// TIA Portal V17 export
// export: Created 2025-03-20T13:42:36.7741063Z, ExportSetting WithDefaults, DisplayName Totally Integrated Automation Portal, DisplayVersion V17 Update 8, DisplayName TIA Portal Openness, DisplayVersion V17 Update 8, DisplayName TIA Portal Version Control Interface, DisplayVersion V17, DisplayName SINAMICS Startdrive Advanced, DisplayVersion V17 SP2, DisplayName SINAMICS Startdrive G110M, G120, G120C, G120D, G120P, G115D, DisplayVersion V17 SP2, DisplayName SINAMICS Startdrive G130, G150, S120, S150, SINAMICS MV, S210, DisplayVersion V17 SP2, DisplayName STEP 7 Professional, DisplayVersion V17 Update 8, DisplayName SINUMERIK ONE STEP 7 Toolbox, DisplayVersion V17 Update 12, DisplayName SINUMERIK 840D sl STEP 7 Toolbox, DisplayVersion V17 Update 12, DisplayName STEP 7 Safety, DisplayVersion V17 Update 6, DisplayName WinCC Advanced, DisplayVersion V17 Update 8
FUNCTION "FC1302_UNIT_03_STATION_0_CYCLE" : Void   // FC1302, LAD
{ S7_Optimized_Access := 'FALSE' }
AUTHOR : ETXETAR
VERSION : 1.0
// stored: AutoNumber false, IsIECCheckEnabled false, SetENOAutomatically false, UDAEnableTagReadback false
   VAR CONSTANT
      FC_NUMBER : DInt := 1302;
   END_VAR
   VAR_TEMP   // added for the SCL form of the ladder/FBD networks
      _w1 : Bool;
   END_VAR
BEGIN

REGION Network 1: GENERAL CONDITIONS
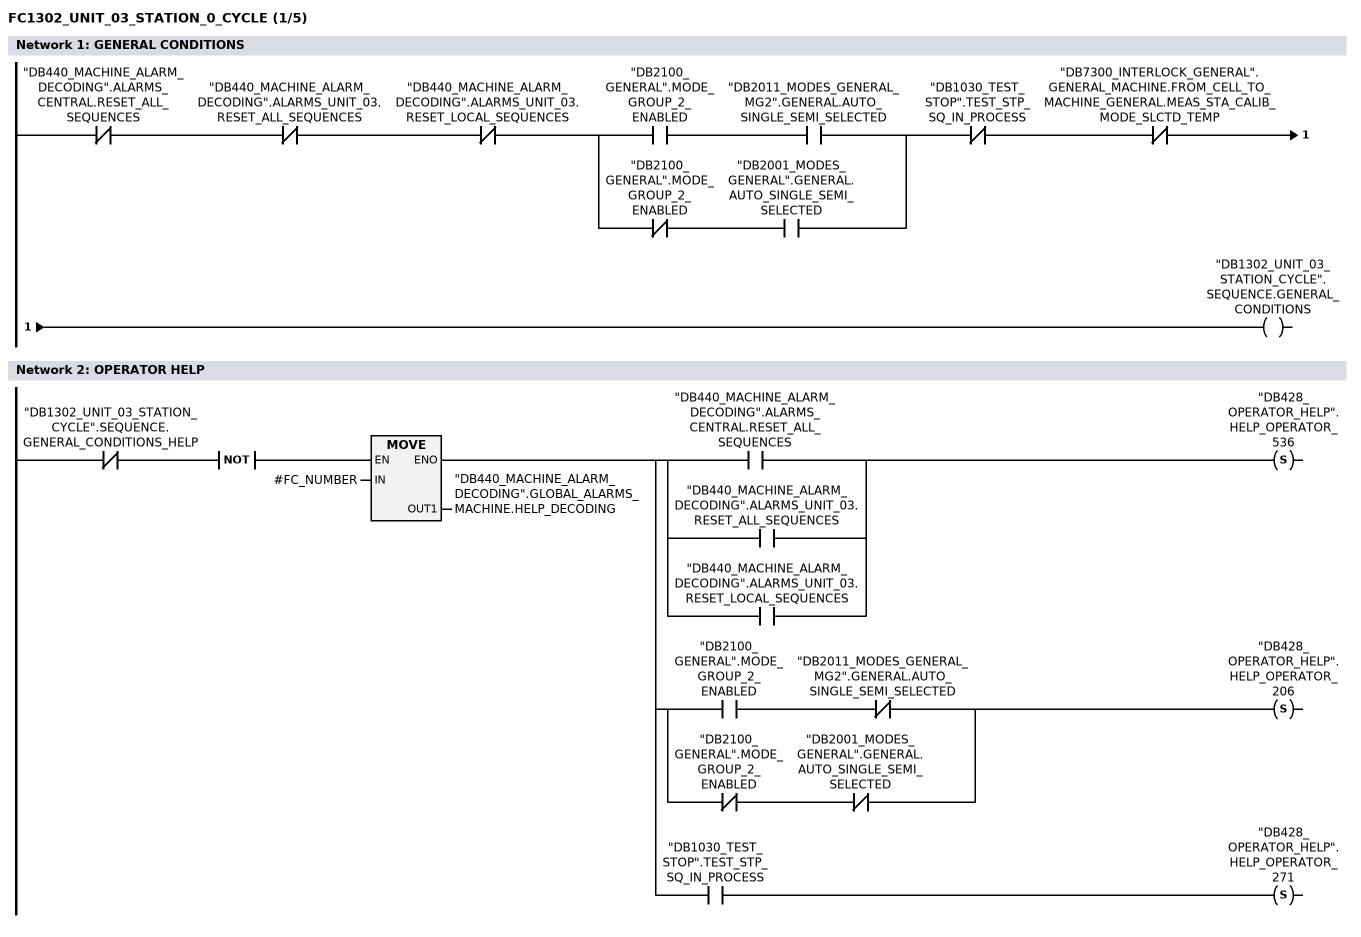
   RUNG wire#powerrail
      I_Contact( "DB440_MACHINE_ALARM_DECODING".ALARMS_CENTRAL.RESET_ALL_SEQUENCES )
      I_Contact( "DB440_MACHINE_ALARM_DECODING".ALARMS_UNIT_03.RESET_ALL_SEQUENCES )
      I_Contact( "DB440_MACHINE_ALARM_DECODING".ALARMS_UNIT_03.RESET_LOCAL_SEQUENCES )
      wire#w1
      Contact( "DB2100_GENERAL".MODE_GROUP_2_ENABLED )
      Contact( "DB2011_MODES_GENERAL_MG2".GENERAL.AUTO_SINGLE_SEMI_SELECTED )
      wire#w2
      I_Contact( "DB1030_TEST_STOP".TEST_STP_SQ_IN_PROCESS )
      I_Contact( "DB7300_INTERLOCK_GENERAL".GENERAL_MACHINE.FROM_CELL_TO_MACHINE_GENERAL.MEAS_STA_CALIB_MODE_SLCTD_TEMP )
      Coil( "DB1302_UNIT_03_STATION_CYCLE".SEQUENCE.GENERAL_CONDITIONS )
   END_RUNG
   RUNG wire#w1
      I_Contact( "DB2100_GENERAL".MODE_GROUP_2_ENABLED )
      Contact( "DB2001_MODES_GENERAL".GENERAL.AUTO_SINGLE_SEMI_SELECTED )
   END_RUNG wire#w2
   // the same network as SCL:
   "DB1302_UNIT_03_STATION_CYCLE".SEQUENCE.GENERAL_CONDITIONS := NOT "DB440_MACHINE_ALARM_DECODING".ALARMS_CENTRAL.RESET_ALL_SEQUENCES AND NOT "DB440_MACHINE_ALARM_DECODING".ALARMS_UNIT_03.RESET_ALL_SEQUENCES AND NOT "DB440_MACHINE_ALARM_DECODING".ALARMS_UNIT_03.RESET_LOCAL_SEQUENCES AND (("DB2100_GENERAL".MODE_GROUP_2_ENABLED AND "DB2011_MODES_GENERAL_MG2".GENERAL.AUTO_SINGLE_SEMI_SELECTED) OR (NOT "DB2100_GENERAL".MODE_GROUP_2_ENABLED AND "DB2001_MODES_GENERAL".GENERAL.AUTO_SINGLE_SEMI_SELECTED)) AND NOT "DB1030_TEST_STOP".TEST_STP_SQ_IN_PROCESS AND NOT "DB7300_INTERLOCK_GENERAL".GENERAL_MACHINE.FROM_CELL_TO_MACHINE_GENERAL.MEAS_STA_CALIB_MODE_SLCTD_TEMP;
END_REGION

REGION Network 2: OPERATOR HELP
   RUNG wire#powerrail
      I_Contact( "DB1302_UNIT_03_STATION_CYCLE".SEQUENCE.GENERAL_CONDITIONS_HELP )
      Not()
      { S7_GenerateENO := "TRUE" } Move(in := #FC_NUMBER, out1 => "DB440_MACHINE_ALARM_DECODING".GLOBAL_ALARMS_MACHINE.HELP_DECODING)
      wire#w1
      Contact( "DB440_MACHINE_ALARM_DECODING".ALARMS_CENTRAL.RESET_ALL_SEQUENCES )
      wire#w2
      S_Coil( "DB428_OPERATOR_HELP".HELP_OPERATOR_536 )
   END_RUNG
   RUNG wire#w1
      Contact( "DB440_MACHINE_ALARM_DECODING".ALARMS_UNIT_03.RESET_ALL_SEQUENCES )
   END_RUNG wire#w2
   RUNG wire#w1
      Contact( "DB440_MACHINE_ALARM_DECODING".ALARMS_UNIT_03.RESET_LOCAL_SEQUENCES )
   END_RUNG wire#w2
   RUNG wire#w1
      Contact( "DB2100_GENERAL".MODE_GROUP_2_ENABLED )
      I_Contact( "DB2011_MODES_GENERAL_MG2".GENERAL.AUTO_SINGLE_SEMI_SELECTED )
      wire#w3
      S_Coil( "DB428_OPERATOR_HELP".HELP_OPERATOR_206 )
   END_RUNG
   RUNG wire#w1
      I_Contact( "DB2100_GENERAL".MODE_GROUP_2_ENABLED )
      I_Contact( "DB2001_MODES_GENERAL".GENERAL.AUTO_SINGLE_SEMI_SELECTED )
   END_RUNG wire#w3
   RUNG wire#w1
      Contact( "DB1030_TEST_STOP".TEST_STP_SQ_IN_PROCESS )
      S_Coil( "DB428_OPERATOR_HELP".HELP_OPERATOR_271 )
   END_RUNG
   // the same network as SCL:
   // ENO of a box is taken as its EN; it also drops when the box reports an error
   #_w1 := NOT (NOT "DB1302_UNIT_03_STATION_CYCLE".SEQUENCE.GENERAL_CONDITIONS_HELP);
   IF #_w1 THEN "DB440_MACHINE_ALARM_DECODING".GLOBAL_ALARMS_MACHINE.HELP_DECODING := #FC_NUMBER; END_IF;
   IF #_w1 AND ("DB440_MACHINE_ALARM_DECODING".ALARMS_CENTRAL.RESET_ALL_SEQUENCES OR "DB440_MACHINE_ALARM_DECODING".ALARMS_UNIT_03.RESET_ALL_SEQUENCES OR "DB440_MACHINE_ALARM_DECODING".ALARMS_UNIT_03.RESET_LOCAL_SEQUENCES) THEN
       "DB428_OPERATOR_HELP".HELP_OPERATOR_536 := TRUE;
   END_IF;
   IF #_w1 AND (("DB2100_GENERAL".MODE_GROUP_2_ENABLED AND NOT "DB2011_MODES_GENERAL_MG2".GENERAL.AUTO_SINGLE_SEMI_SELECTED) OR (NOT "DB2100_GENERAL".MODE_GROUP_2_ENABLED AND NOT "DB2001_MODES_GENERAL".GENERAL.AUTO_SINGLE_SEMI_SELECTED)) THEN
       "DB428_OPERATOR_HELP".HELP_OPERATOR_206 := TRUE;
   END_IF;
   IF #_w1 AND "DB1030_TEST_STOP".TEST_STP_SQ_IN_PROCESS THEN
       "DB428_OPERATOR_HELP".HELP_OPERATOR_271 := TRUE;
   END_IF;
END_REGION

REGION Network 3: INITIAL CONDITIONS
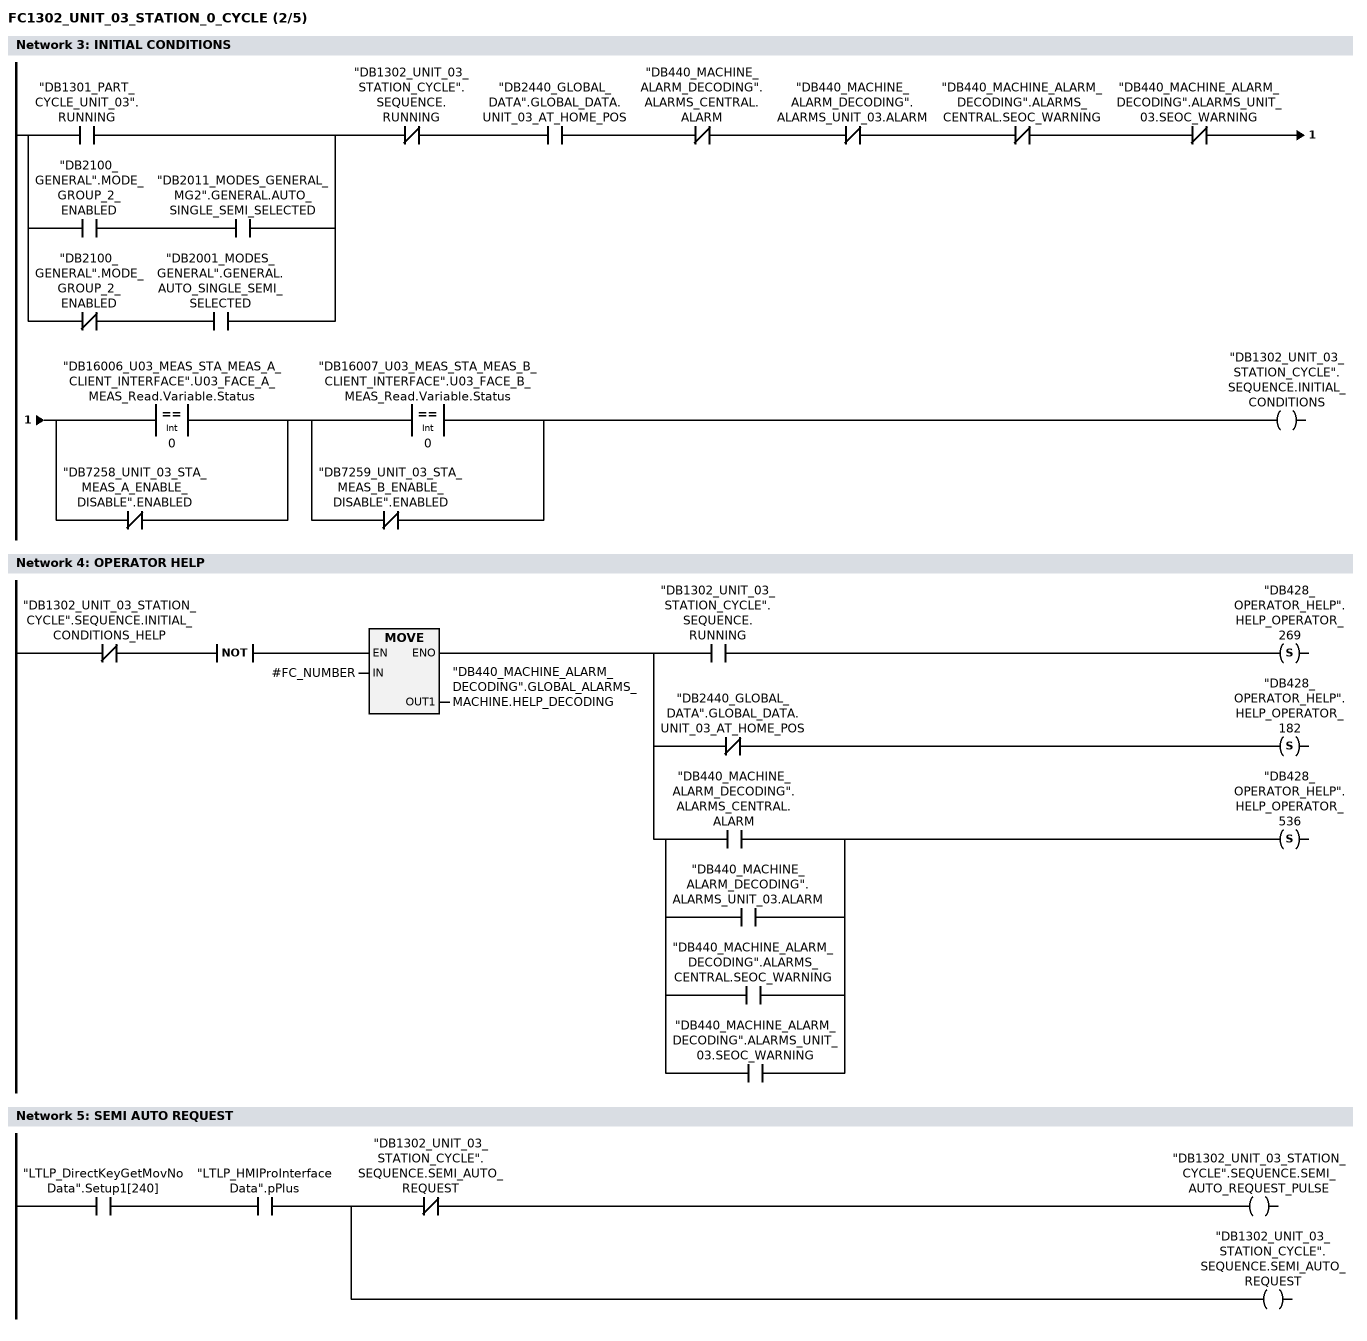
   RUNG wire#powerrail
      Contact( "DB1301_PART_CYCLE_UNIT_03".RUNNING )
      wire#w1
      I_Contact( "DB1302_UNIT_03_STATION_CYCLE".SEQUENCE.RUNNING )
      Contact( "DB2440_GLOBAL_DATA".GLOBAL_DATA.UNIT_03_AT_HOME_POS )
      I_Contact( "DB440_MACHINE_ALARM_DECODING".ALARMS_CENTRAL.ALARM )
      I_Contact( "DB440_MACHINE_ALARM_DECODING".ALARMS_UNIT_03.ALARM )
      I_Contact( "DB440_MACHINE_ALARM_DECODING".ALARMS_CENTRAL.SEOC_WARNING )
      I_Contact( "DB440_MACHINE_ALARM_DECODING".ALARMS_UNIT_03.SEOC_WARNING )
      wire#w2
      { S7_Templates := "SrcType := Int" } EQ_Contact(in1 := "DB16006_U03_MEAS_STA_MEAS_A_CLIENT_INTERFACE".U03_FACE_A_MEAS_Read.Variable.Status, in2 := 0)
      wire#w3
      { S7_Templates := "SrcType := Int" } EQ_Contact(in1 := "DB16007_U03_MEAS_STA_MEAS_B_CLIENT_INTERFACE".U03_FACE_B_MEAS_Read.Variable.Status, in2 := 0)
      wire#w4
      Coil( "DB1302_UNIT_03_STATION_CYCLE".SEQUENCE.INITIAL_CONDITIONS )
   END_RUNG
   RUNG wire#powerrail
      Contact( "DB2100_GENERAL".MODE_GROUP_2_ENABLED )
      Contact( "DB2011_MODES_GENERAL_MG2".GENERAL.AUTO_SINGLE_SEMI_SELECTED )
   END_RUNG wire#w1
   RUNG wire#powerrail
      I_Contact( "DB2100_GENERAL".MODE_GROUP_2_ENABLED )
      Contact( "DB2001_MODES_GENERAL".GENERAL.AUTO_SINGLE_SEMI_SELECTED )
   END_RUNG wire#w1
   RUNG wire#w2
      I_Contact( "DB7258_UNIT_03_STA_MEAS_A_ENABLE_DISABLE".ENABLED )
   END_RUNG wire#w3
   RUNG wire#w3
      I_Contact( "DB7259_UNIT_03_STA_MEAS_B_ENABLE_DISABLE".ENABLED )
   END_RUNG wire#w4
   // the same network as SCL:
   "DB1302_UNIT_03_STATION_CYCLE".SEQUENCE.INITIAL_CONDITIONS := ("DB1301_PART_CYCLE_UNIT_03".RUNNING OR ("DB2100_GENERAL".MODE_GROUP_2_ENABLED AND "DB2011_MODES_GENERAL_MG2".GENERAL.AUTO_SINGLE_SEMI_SELECTED) OR (NOT "DB2100_GENERAL".MODE_GROUP_2_ENABLED AND "DB2001_MODES_GENERAL".GENERAL.AUTO_SINGLE_SEMI_SELECTED)) AND NOT "DB1302_UNIT_03_STATION_CYCLE".SEQUENCE.RUNNING AND "DB2440_GLOBAL_DATA".GLOBAL_DATA.UNIT_03_AT_HOME_POS AND NOT "DB440_MACHINE_ALARM_DECODING".ALARMS_CENTRAL.ALARM AND NOT "DB440_MACHINE_ALARM_DECODING".ALARMS_UNIT_03.ALARM AND NOT "DB440_MACHINE_ALARM_DECODING".ALARMS_CENTRAL.SEOC_WARNING AND NOT "DB440_MACHINE_ALARM_DECODING".ALARMS_UNIT_03.SEOC_WARNING AND (("DB16006_U03_MEAS_STA_MEAS_A_CLIENT_INTERFACE".U03_FACE_A_MEAS_Read.Variable.Status = 0) OR NOT "DB7258_UNIT_03_STA_MEAS_A_ENABLE_DISABLE".ENABLED) AND (("DB16007_U03_MEAS_STA_MEAS_B_CLIENT_INTERFACE".U03_FACE_B_MEAS_Read.Variable.Status = 0) OR NOT "DB7259_UNIT_03_STA_MEAS_B_ENABLE_DISABLE".ENABLED);
END_REGION

REGION Network 4: OPERATOR HELP
   RUNG wire#powerrail
      I_Contact( "DB1302_UNIT_03_STATION_CYCLE".SEQUENCE.INITIAL_CONDITIONS_HELP )
      Not()
      { S7_GenerateENO := "TRUE" } Move(in := #FC_NUMBER, out1 => "DB440_MACHINE_ALARM_DECODING".GLOBAL_ALARMS_MACHINE.HELP_DECODING)
      wire#w1
      Contact( "DB1302_UNIT_03_STATION_CYCLE".SEQUENCE.RUNNING )
      S_Coil( "DB428_OPERATOR_HELP".HELP_OPERATOR_269 )
   END_RUNG
   RUNG wire#w1
      I_Contact( "DB2440_GLOBAL_DATA".GLOBAL_DATA.UNIT_03_AT_HOME_POS )
      S_Coil( "DB428_OPERATOR_HELP".HELP_OPERATOR_182 )
   END_RUNG
   RUNG wire#w1
      Contact( "DB440_MACHINE_ALARM_DECODING".ALARMS_CENTRAL.ALARM )
      wire#w2
      S_Coil( "DB428_OPERATOR_HELP".HELP_OPERATOR_536 )
   END_RUNG
   RUNG wire#w1
      Contact( "DB440_MACHINE_ALARM_DECODING".ALARMS_UNIT_03.ALARM )
   END_RUNG wire#w2
   RUNG wire#w1
      Contact( "DB440_MACHINE_ALARM_DECODING".ALARMS_CENTRAL.SEOC_WARNING )
   END_RUNG wire#w2
   RUNG wire#w1
      Contact( "DB440_MACHINE_ALARM_DECODING".ALARMS_UNIT_03.SEOC_WARNING )
   END_RUNG wire#w2
   // the same network as SCL:
   // ENO of a box is taken as its EN; it also drops when the box reports an error
   #_w1 := NOT (NOT "DB1302_UNIT_03_STATION_CYCLE".SEQUENCE.INITIAL_CONDITIONS_HELP);
   IF #_w1 THEN "DB440_MACHINE_ALARM_DECODING".GLOBAL_ALARMS_MACHINE.HELP_DECODING := #FC_NUMBER; END_IF;
   IF #_w1 AND "DB1302_UNIT_03_STATION_CYCLE".SEQUENCE.RUNNING THEN
       "DB428_OPERATOR_HELP".HELP_OPERATOR_269 := TRUE;
   END_IF;
   IF #_w1 AND NOT "DB2440_GLOBAL_DATA".GLOBAL_DATA.UNIT_03_AT_HOME_POS THEN
       "DB428_OPERATOR_HELP".HELP_OPERATOR_182 := TRUE;
   END_IF;
   IF #_w1 AND ("DB440_MACHINE_ALARM_DECODING".ALARMS_CENTRAL.ALARM OR "DB440_MACHINE_ALARM_DECODING".ALARMS_UNIT_03.ALARM OR "DB440_MACHINE_ALARM_DECODING".ALARMS_CENTRAL.SEOC_WARNING OR "DB440_MACHINE_ALARM_DECODING".ALARMS_UNIT_03.SEOC_WARNING) THEN
       "DB428_OPERATOR_HELP".HELP_OPERATOR_536 := TRUE;
   END_IF;
END_REGION

REGION Network 5: SEMI AUTO REQUEST
   RUNG wire#powerrail
      Contact( "LTLP_DirectKeyGetMovNoData".Setup1[240] )
      Contact( "LTLP_HMIProInterfaceData".pPlus )
      wire#w1
      I_Contact( "DB1302_UNIT_03_STATION_CYCLE".SEQUENCE.SEMI_AUTO_REQUEST )
      Coil( "DB1302_UNIT_03_STATION_CYCLE".SEQUENCE.SEMI_AUTO_REQUEST_PULSE )
   END_RUNG
   RUNG wire#w1
      Coil( "DB1302_UNIT_03_STATION_CYCLE".SEQUENCE.SEMI_AUTO_REQUEST )
   END_RUNG
   // the same network as SCL:
   #_w1 := "LTLP_DirectKeyGetMovNoData".Setup1[240] AND "LTLP_HMIProInterfaceData".pPlus;
   "DB1302_UNIT_03_STATION_CYCLE".SEQUENCE.SEMI_AUTO_REQUEST_PULSE := #_w1 AND NOT "DB1302_UNIT_03_STATION_CYCLE".SEQUENCE.SEMI_AUTO_REQUEST;
   "DB1302_UNIT_03_STATION_CYCLE".SEQUENCE.SEMI_AUTO_REQUEST := #_w1;
END_REGION

REGION Network 6: OPERATOR HELP
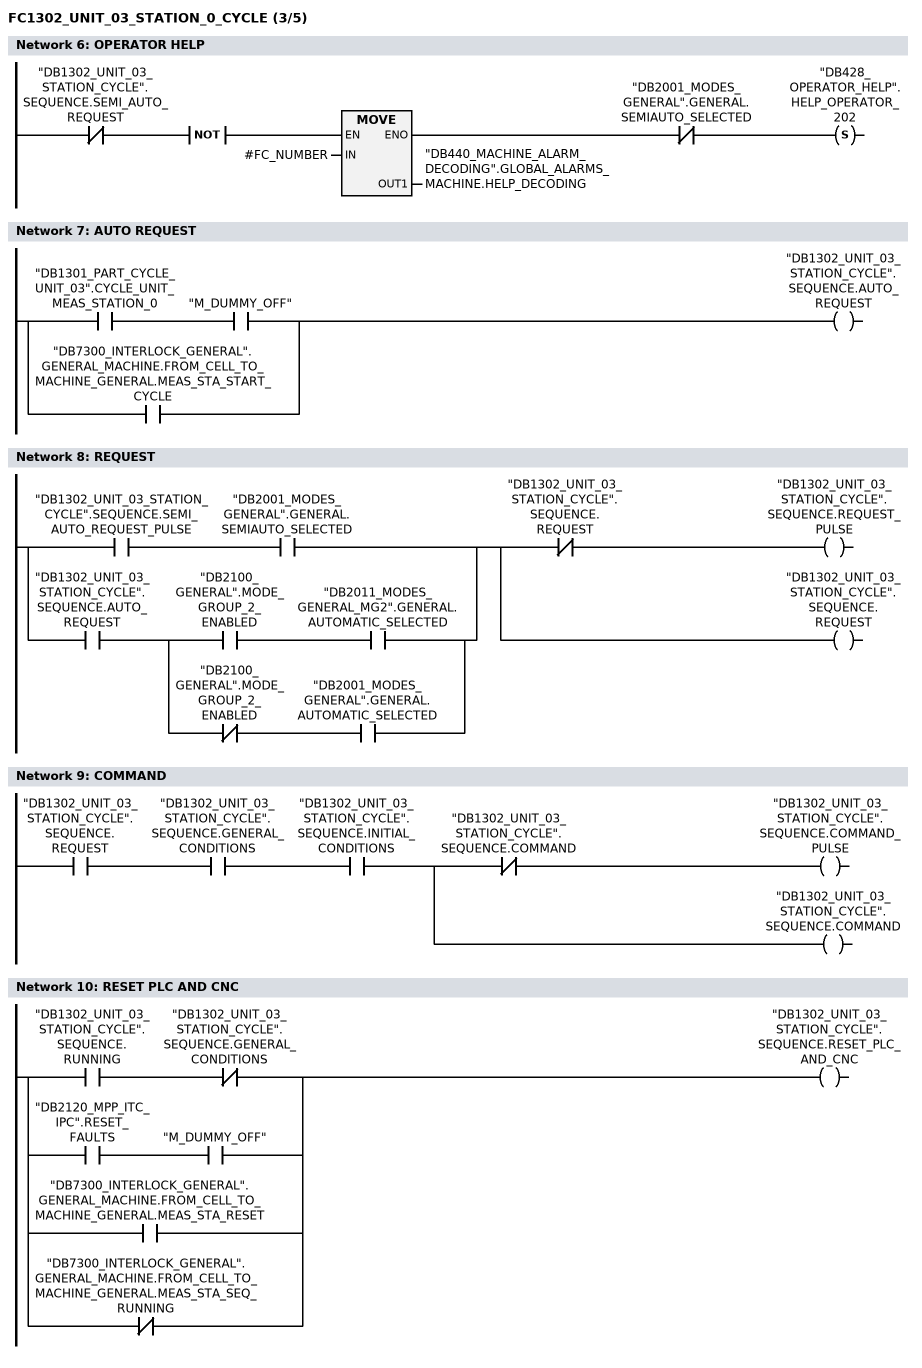
   RUNG wire#powerrail
      I_Contact( "DB1302_UNIT_03_STATION_CYCLE".SEQUENCE.SEMI_AUTO_REQUEST )
      Not()
      { S7_GenerateENO := "TRUE" } Move(in := #FC_NUMBER, out1 => "DB440_MACHINE_ALARM_DECODING".GLOBAL_ALARMS_MACHINE.HELP_DECODING)
      I_Contact( "DB2001_MODES_GENERAL".GENERAL.SEMIAUTO_SELECTED )
      S_Coil( "DB428_OPERATOR_HELP".HELP_OPERATOR_202 )
   END_RUNG
   // the same network as SCL:
   // ENO of a box is taken as its EN; it also drops when the box reports an error
   #_w1 := NOT (NOT "DB1302_UNIT_03_STATION_CYCLE".SEQUENCE.SEMI_AUTO_REQUEST);
   IF #_w1 THEN "DB440_MACHINE_ALARM_DECODING".GLOBAL_ALARMS_MACHINE.HELP_DECODING := #FC_NUMBER; END_IF;
   IF #_w1 AND NOT "DB2001_MODES_GENERAL".GENERAL.SEMIAUTO_SELECTED THEN
       "DB428_OPERATOR_HELP".HELP_OPERATOR_202 := TRUE;
   END_IF;
END_REGION

REGION Network 7: AUTO REQUEST
   RUNG wire#powerrail
      Contact( "DB1301_PART_CYCLE_UNIT_03".CYCLE_UNIT_MEAS_STATION_0 )
      Contact( "M_DUMMY_OFF" )
      wire#w1
      Coil( "DB1302_UNIT_03_STATION_CYCLE".SEQUENCE.AUTO_REQUEST )
   END_RUNG
   RUNG wire#powerrail
      Contact( "DB7300_INTERLOCK_GENERAL".GENERAL_MACHINE.FROM_CELL_TO_MACHINE_GENERAL.MEAS_STA_START_CYCLE )
   END_RUNG wire#w1
   // the same network as SCL:
   "DB1302_UNIT_03_STATION_CYCLE".SEQUENCE.AUTO_REQUEST := ("DB1301_PART_CYCLE_UNIT_03".CYCLE_UNIT_MEAS_STATION_0 AND "M_DUMMY_OFF") OR "DB7300_INTERLOCK_GENERAL".GENERAL_MACHINE.FROM_CELL_TO_MACHINE_GENERAL.MEAS_STA_START_CYCLE;
END_REGION

REGION Network 8: REQUEST
   RUNG wire#powerrail
      Contact( "DB1302_UNIT_03_STATION_CYCLE".SEQUENCE.SEMI_AUTO_REQUEST_PULSE )
      Contact( "DB2001_MODES_GENERAL".GENERAL.SEMIAUTO_SELECTED )
      wire#w1
      I_Contact( "DB1302_UNIT_03_STATION_CYCLE".SEQUENCE.REQUEST )
      Coil( "DB1302_UNIT_03_STATION_CYCLE".SEQUENCE.REQUEST_PULSE )
   END_RUNG
   RUNG wire#powerrail
      Contact( "DB1302_UNIT_03_STATION_CYCLE".SEQUENCE.AUTO_REQUEST )
      wire#w2
      Contact( "DB2100_GENERAL".MODE_GROUP_2_ENABLED )
      Contact( "DB2011_MODES_GENERAL_MG2".GENERAL.AUTOMATIC_SELECTED )
   END_RUNG wire#w1
   RUNG wire#w2
      I_Contact( "DB2100_GENERAL".MODE_GROUP_2_ENABLED )
      Contact( "DB2001_MODES_GENERAL".GENERAL.AUTOMATIC_SELECTED )
   END_RUNG wire#w1
   RUNG wire#w1
      Coil( "DB1302_UNIT_03_STATION_CYCLE".SEQUENCE.REQUEST )
   END_RUNG
   // the same network as SCL:
   #_w1 := ("DB1302_UNIT_03_STATION_CYCLE".SEQUENCE.SEMI_AUTO_REQUEST_PULSE AND "DB2001_MODES_GENERAL".GENERAL.SEMIAUTO_SELECTED) OR ("DB1302_UNIT_03_STATION_CYCLE".SEQUENCE.AUTO_REQUEST AND (("DB2100_GENERAL".MODE_GROUP_2_ENABLED AND "DB2011_MODES_GENERAL_MG2".GENERAL.AUTOMATIC_SELECTED) OR (NOT "DB2100_GENERAL".MODE_GROUP_2_ENABLED AND "DB2001_MODES_GENERAL".GENERAL.AUTOMATIC_SELECTED)));
   "DB1302_UNIT_03_STATION_CYCLE".SEQUENCE.REQUEST_PULSE := #_w1 AND NOT "DB1302_UNIT_03_STATION_CYCLE".SEQUENCE.REQUEST;
   "DB1302_UNIT_03_STATION_CYCLE".SEQUENCE.REQUEST := #_w1;
END_REGION

REGION Network 9: COMMAND
   RUNG wire#powerrail
      Contact( "DB1302_UNIT_03_STATION_CYCLE".SEQUENCE.REQUEST )
      Contact( "DB1302_UNIT_03_STATION_CYCLE".SEQUENCE.GENERAL_CONDITIONS )
      Contact( "DB1302_UNIT_03_STATION_CYCLE".SEQUENCE.INITIAL_CONDITIONS )
      wire#w1
      I_Contact( "DB1302_UNIT_03_STATION_CYCLE".SEQUENCE.COMMAND )
      Coil( "DB1302_UNIT_03_STATION_CYCLE".SEQUENCE.COMMAND_PULSE )
   END_RUNG
   RUNG wire#w1
      Coil( "DB1302_UNIT_03_STATION_CYCLE".SEQUENCE.COMMAND )
   END_RUNG
   // the same network as SCL:
   #_w1 := "DB1302_UNIT_03_STATION_CYCLE".SEQUENCE.REQUEST AND "DB1302_UNIT_03_STATION_CYCLE".SEQUENCE.GENERAL_CONDITIONS AND "DB1302_UNIT_03_STATION_CYCLE".SEQUENCE.INITIAL_CONDITIONS;
   "DB1302_UNIT_03_STATION_CYCLE".SEQUENCE.COMMAND_PULSE := #_w1 AND NOT "DB1302_UNIT_03_STATION_CYCLE".SEQUENCE.COMMAND;
   "DB1302_UNIT_03_STATION_CYCLE".SEQUENCE.COMMAND := #_w1;
END_REGION

REGION Network 10: RESET PLC AND CNC
   RUNG wire#powerrail
      Contact( "DB1302_UNIT_03_STATION_CYCLE".SEQUENCE.RUNNING )
      I_Contact( "DB1302_UNIT_03_STATION_CYCLE".SEQUENCE.GENERAL_CONDITIONS )
      wire#w1
      Coil( "DB1302_UNIT_03_STATION_CYCLE".SEQUENCE.RESET_PLC_AND_CNC )
   END_RUNG
   RUNG wire#powerrail
      Contact( "DB2120_MPP_ITC_IPC".RESET_FAULTS )
      Contact( "M_DUMMY_OFF" )
   END_RUNG wire#w1
   RUNG wire#powerrail
      Contact( "DB7300_INTERLOCK_GENERAL".GENERAL_MACHINE.FROM_CELL_TO_MACHINE_GENERAL.MEAS_STA_RESET )
   END_RUNG wire#w1
   RUNG wire#powerrail
      I_Contact( "DB7300_INTERLOCK_GENERAL".GENERAL_MACHINE.FROM_CELL_TO_MACHINE_GENERAL.MEAS_STA_SEQ_RUNNING )
   END_RUNG wire#w1
   // the same network as SCL:
   "DB1302_UNIT_03_STATION_CYCLE".SEQUENCE.RESET_PLC_AND_CNC := ("DB1302_UNIT_03_STATION_CYCLE".SEQUENCE.RUNNING AND NOT "DB1302_UNIT_03_STATION_CYCLE".SEQUENCE.GENERAL_CONDITIONS) OR ("DB2120_MPP_ITC_IPC".RESET_FAULTS AND "M_DUMMY_OFF") OR "DB7300_INTERLOCK_GENERAL".GENERAL_MACHINE.FROM_CELL_TO_MACHINE_GENERAL.MEAS_STA_RESET OR NOT "DB7300_INTERLOCK_GENERAL".GENERAL_MACHINE.FROM_CELL_TO_MACHINE_GENERAL.MEAS_STA_SEQ_RUNNING;
END_REGION

REGION Network 11: RUNNING
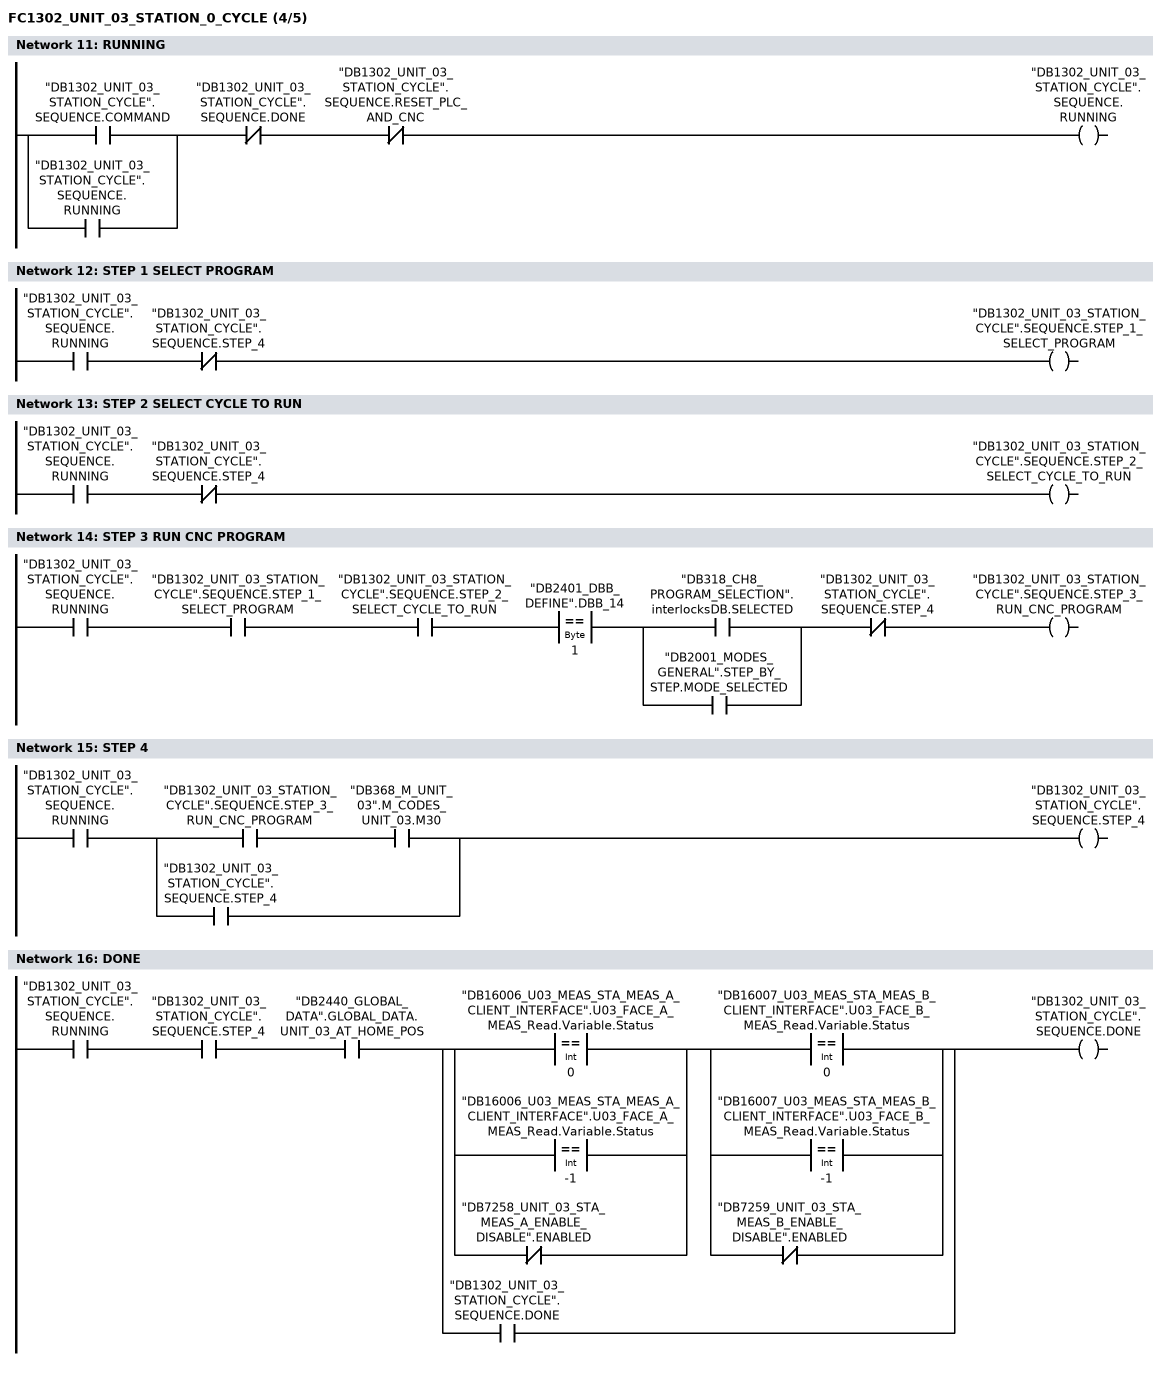
   RUNG wire#powerrail
      Contact( "DB1302_UNIT_03_STATION_CYCLE".SEQUENCE.COMMAND )
      wire#w1
      I_Contact( "DB1302_UNIT_03_STATION_CYCLE".SEQUENCE.DONE )
      I_Contact( "DB1302_UNIT_03_STATION_CYCLE".SEQUENCE.RESET_PLC_AND_CNC )
      Coil( "DB1302_UNIT_03_STATION_CYCLE".SEQUENCE.RUNNING )
   END_RUNG
   RUNG wire#powerrail
      Contact( "DB1302_UNIT_03_STATION_CYCLE".SEQUENCE.RUNNING )
   END_RUNG wire#w1
   // the same network as SCL:
   "DB1302_UNIT_03_STATION_CYCLE".SEQUENCE.RUNNING := ("DB1302_UNIT_03_STATION_CYCLE".SEQUENCE.COMMAND OR "DB1302_UNIT_03_STATION_CYCLE".SEQUENCE.RUNNING) AND NOT "DB1302_UNIT_03_STATION_CYCLE".SEQUENCE.DONE AND NOT "DB1302_UNIT_03_STATION_CYCLE".SEQUENCE.RESET_PLC_AND_CNC;
END_REGION

REGION Network 12: STEP 1 SELECT PROGRAM
   RUNG wire#powerrail
      Contact( "DB1302_UNIT_03_STATION_CYCLE".SEQUENCE.RUNNING )
      I_Contact( "DB1302_UNIT_03_STATION_CYCLE".SEQUENCE.STEP_4 )
      Coil( "DB1302_UNIT_03_STATION_CYCLE".SEQUENCE.STEP_1_SELECT_PROGRAM )
   END_RUNG
   // the same network as SCL:
   "DB1302_UNIT_03_STATION_CYCLE".SEQUENCE.STEP_1_SELECT_PROGRAM := "DB1302_UNIT_03_STATION_CYCLE".SEQUENCE.RUNNING AND NOT "DB1302_UNIT_03_STATION_CYCLE".SEQUENCE.STEP_4;
END_REGION

REGION Network 13: STEP 2 SELECT CYCLE TO RUN
   RUNG wire#powerrail
      Contact( "DB1302_UNIT_03_STATION_CYCLE".SEQUENCE.RUNNING )
      I_Contact( "DB1302_UNIT_03_STATION_CYCLE".SEQUENCE.STEP_4 )
      Coil( "DB1302_UNIT_03_STATION_CYCLE".SEQUENCE.STEP_2_SELECT_CYCLE_TO_RUN )
   END_RUNG
   // the same network as SCL:
   "DB1302_UNIT_03_STATION_CYCLE".SEQUENCE.STEP_2_SELECT_CYCLE_TO_RUN := "DB1302_UNIT_03_STATION_CYCLE".SEQUENCE.RUNNING AND NOT "DB1302_UNIT_03_STATION_CYCLE".SEQUENCE.STEP_4;
END_REGION

REGION Network 14: STEP 3 RUN CNC PROGRAM
   RUNG wire#powerrail
      Contact( "DB1302_UNIT_03_STATION_CYCLE".SEQUENCE.RUNNING )
      Contact( "DB1302_UNIT_03_STATION_CYCLE".SEQUENCE.STEP_1_SELECT_PROGRAM )
      Contact( "DB1302_UNIT_03_STATION_CYCLE".SEQUENCE.STEP_2_SELECT_CYCLE_TO_RUN )
      { S7_Templates := "SrcType := Byte" } EQ_Contact(in1 := "DB2401_DBB_DEFINE".DBB_14, in2 := 1)
      wire#w1
      Contact( "DB318_CH8_PROGRAM_SELECTION".interlocksDB.SELECTED )
      wire#w2
      I_Contact( "DB1302_UNIT_03_STATION_CYCLE".SEQUENCE.STEP_4 )
      Coil( "DB1302_UNIT_03_STATION_CYCLE".SEQUENCE.STEP_3_RUN_CNC_PROGRAM )
   END_RUNG
   RUNG wire#w1
      Contact( "DB2001_MODES_GENERAL".STEP_BY_STEP.MODE_SELECTED )
   END_RUNG wire#w2
   // the same network as SCL:
   "DB1302_UNIT_03_STATION_CYCLE".SEQUENCE.STEP_3_RUN_CNC_PROGRAM := "DB1302_UNIT_03_STATION_CYCLE".SEQUENCE.RUNNING AND "DB1302_UNIT_03_STATION_CYCLE".SEQUENCE.STEP_1_SELECT_PROGRAM AND "DB1302_UNIT_03_STATION_CYCLE".SEQUENCE.STEP_2_SELECT_CYCLE_TO_RUN AND ("DB2401_DBB_DEFINE".DBB_14 = 1) AND ("DB318_CH8_PROGRAM_SELECTION".interlocksDB.SELECTED OR "DB2001_MODES_GENERAL".STEP_BY_STEP.MODE_SELECTED) AND NOT "DB1302_UNIT_03_STATION_CYCLE".SEQUENCE.STEP_4;
END_REGION

REGION Network 15: STEP 4
   RUNG wire#powerrail
      Contact( "DB1302_UNIT_03_STATION_CYCLE".SEQUENCE.RUNNING )
      wire#w1
      Contact( "DB1302_UNIT_03_STATION_CYCLE".SEQUENCE.STEP_3_RUN_CNC_PROGRAM )
      Contact( "DB368_M_UNIT_03".M_CODES_UNIT_03.M30 )
      wire#w2
      Coil( "DB1302_UNIT_03_STATION_CYCLE".SEQUENCE.STEP_4 )
   END_RUNG
   RUNG wire#w1
      Contact( "DB1302_UNIT_03_STATION_CYCLE".SEQUENCE.STEP_4 )
   END_RUNG wire#w2
   // the same network as SCL:
   "DB1302_UNIT_03_STATION_CYCLE".SEQUENCE.STEP_4 := "DB1302_UNIT_03_STATION_CYCLE".SEQUENCE.RUNNING AND (("DB1302_UNIT_03_STATION_CYCLE".SEQUENCE.STEP_3_RUN_CNC_PROGRAM AND "DB368_M_UNIT_03".M_CODES_UNIT_03.M30) OR "DB1302_UNIT_03_STATION_CYCLE".SEQUENCE.STEP_4);
END_REGION

REGION Network 16: DONE
   RUNG wire#powerrail
      Contact( "DB1302_UNIT_03_STATION_CYCLE".SEQUENCE.RUNNING )
      Contact( "DB1302_UNIT_03_STATION_CYCLE".SEQUENCE.STEP_4 )
      Contact( "DB2440_GLOBAL_DATA".GLOBAL_DATA.UNIT_03_AT_HOME_POS )
      wire#w1
      { S7_Templates := "SrcType := Int" } EQ_Contact(in1 := "DB16006_U03_MEAS_STA_MEAS_A_CLIENT_INTERFACE".U03_FACE_A_MEAS_Read.Variable.Status, in2 := 0)
      wire#w2
      { S7_Templates := "SrcType := Int" } EQ_Contact(in1 := "DB16007_U03_MEAS_STA_MEAS_B_CLIENT_INTERFACE".U03_FACE_B_MEAS_Read.Variable.Status, in2 := 0)
      wire#w3
      Coil( "DB1302_UNIT_03_STATION_CYCLE".SEQUENCE.DONE )
   END_RUNG
   RUNG wire#w1
      { S7_Templates := "SrcType := Int" } EQ_Contact(in1 := "DB16006_U03_MEAS_STA_MEAS_A_CLIENT_INTERFACE".U03_FACE_A_MEAS_Read.Variable.Status, in2 := -1)
   END_RUNG wire#w2
   RUNG wire#w1
      I_Contact( "DB7258_UNIT_03_STA_MEAS_A_ENABLE_DISABLE".ENABLED )
   END_RUNG wire#w2
   RUNG wire#w2
      { S7_Templates := "SrcType := Int" } EQ_Contact(in1 := "DB16007_U03_MEAS_STA_MEAS_B_CLIENT_INTERFACE".U03_FACE_B_MEAS_Read.Variable.Status, in2 := -1)
   END_RUNG wire#w3
   RUNG wire#w2
      I_Contact( "DB7259_UNIT_03_STA_MEAS_B_ENABLE_DISABLE".ENABLED )
   END_RUNG wire#w3
   RUNG wire#w1
      Contact( "DB1302_UNIT_03_STATION_CYCLE".SEQUENCE.DONE )
   END_RUNG wire#w3
   // the same network as SCL:
   "DB1302_UNIT_03_STATION_CYCLE".SEQUENCE.DONE := "DB1302_UNIT_03_STATION_CYCLE".SEQUENCE.RUNNING AND "DB1302_UNIT_03_STATION_CYCLE".SEQUENCE.STEP_4 AND "DB2440_GLOBAL_DATA".GLOBAL_DATA.UNIT_03_AT_HOME_POS AND (((("DB16006_U03_MEAS_STA_MEAS_A_CLIENT_INTERFACE".U03_FACE_A_MEAS_Read.Variable.Status = 0) OR ("DB16006_U03_MEAS_STA_MEAS_A_CLIENT_INTERFACE".U03_FACE_A_MEAS_Read.Variable.Status = (-1)) OR NOT "DB7258_UNIT_03_STA_MEAS_A_ENABLE_DISABLE".ENABLED) AND (("DB16007_U03_MEAS_STA_MEAS_B_CLIENT_INTERFACE".U03_FACE_B_MEAS_Read.Variable.Status = 0) OR ("DB16007_U03_MEAS_STA_MEAS_B_CLIENT_INTERFACE".U03_FACE_B_MEAS_Read.Variable.Status = (-1)) OR NOT "DB7259_UNIT_03_STA_MEAS_B_ENABLE_DISABLE".ENABLED)) OR "DB1302_UNIT_03_STATION_CYCLE".SEQUENCE.DONE);
END_REGION

REGION Network 17: TIME EXCEEDED ALARM
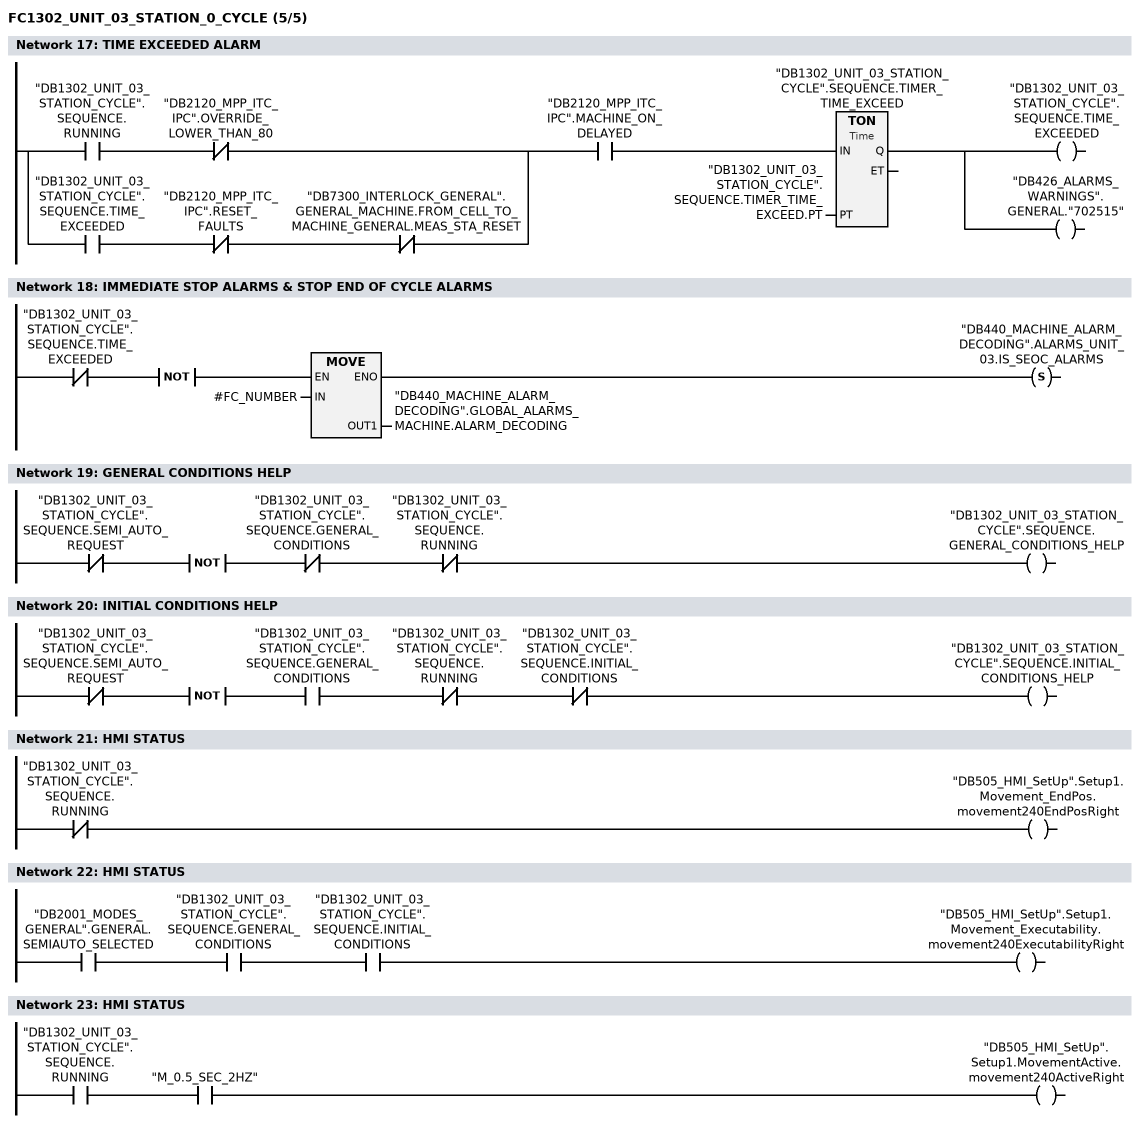
   RUNG wire#powerrail
      Contact( "DB1302_UNIT_03_STATION_CYCLE".SEQUENCE.RUNNING )
      I_Contact( "DB2120_MPP_ITC_IPC".OVERRIDE_LOWER_THAN_80 )
      wire#w1
      Contact( "DB2120_MPP_ITC_IPC".MACHINE_ON_DELAYED )
      { S7_Templates := "time_type := Time" } "DB1302_UNIT_03_STATION_CYCLE".SEQUENCE.TIMER_TIME_EXCEED.TON(pt := "DB1302_UNIT_03_STATION_CYCLE".SEQUENCE.TIMER_TIME_EXCEED.PT, et =>)
      wire#w2
      Coil( "DB1302_UNIT_03_STATION_CYCLE".SEQUENCE.TIME_EXCEEDED )
   END_RUNG
   RUNG wire#powerrail
      Contact( "DB1302_UNIT_03_STATION_CYCLE".SEQUENCE.TIME_EXCEEDED )
      I_Contact( "DB2120_MPP_ITC_IPC".RESET_FAULTS )
      I_Contact( "DB7300_INTERLOCK_GENERAL".GENERAL_MACHINE.FROM_CELL_TO_MACHINE_GENERAL.MEAS_STA_RESET )
   END_RUNG wire#w1
   RUNG wire#w2
      Coil( "DB426_ALARMS_WARNINGS".GENERAL."702515" )
   END_RUNG
   // the same network as SCL:
   "DB1302_UNIT_03_STATION_CYCLE".SEQUENCE.TIMER_TIME_EXCEED.TON(IN := (("DB1302_UNIT_03_STATION_CYCLE".SEQUENCE.RUNNING AND NOT "DB2120_MPP_ITC_IPC".OVERRIDE_LOWER_THAN_80) OR ("DB1302_UNIT_03_STATION_CYCLE".SEQUENCE.TIME_EXCEEDED AND NOT "DB2120_MPP_ITC_IPC".RESET_FAULTS AND NOT "DB7300_INTERLOCK_GENERAL".GENERAL_MACHINE.FROM_CELL_TO_MACHINE_GENERAL.MEAS_STA_RESET)) AND "DB2120_MPP_ITC_IPC".MACHINE_ON_DELAYED,
                           PT := "DB1302_UNIT_03_STATION_CYCLE".SEQUENCE.TIMER_TIME_EXCEED.PT);
   "DB1302_UNIT_03_STATION_CYCLE".SEQUENCE.TIME_EXCEEDED := "DB1302_UNIT_03_STATION_CYCLE".SEQUENCE.TIMER_TIME_EXCEED.Q;
   "DB426_ALARMS_WARNINGS".GENERAL."702515" := "DB1302_UNIT_03_STATION_CYCLE".SEQUENCE.TIMER_TIME_EXCEED.Q;
END_REGION

REGION Network 18: IMMEDIATE STOP ALARMS & STOP END OF CYCLE ALARMS
   RUNG wire#powerrail
      I_Contact( "DB1302_UNIT_03_STATION_CYCLE".SEQUENCE.TIME_EXCEEDED )
      Not()
      { S7_GenerateENO := "TRUE" } Move(in := #FC_NUMBER, out1 => "DB440_MACHINE_ALARM_DECODING".GLOBAL_ALARMS_MACHINE.ALARM_DECODING)
      S_Coil( "DB440_MACHINE_ALARM_DECODING".ALARMS_UNIT_03.IS_SEOC_ALARMS )
   END_RUNG
   // the same network as SCL:
   // ENO of a box is taken as its EN; it also drops when the box reports an error
   IF NOT (NOT "DB1302_UNIT_03_STATION_CYCLE".SEQUENCE.TIME_EXCEEDED) THEN
       "DB440_MACHINE_ALARM_DECODING".GLOBAL_ALARMS_MACHINE.ALARM_DECODING := #FC_NUMBER;
       "DB440_MACHINE_ALARM_DECODING".ALARMS_UNIT_03.IS_SEOC_ALARMS := TRUE;
   END_IF;
END_REGION

REGION Network 19: GENERAL CONDITIONS HELP
   RUNG wire#powerrail
      I_Contact( "DB1302_UNIT_03_STATION_CYCLE".SEQUENCE.SEMI_AUTO_REQUEST )
      Not()
      I_Contact( "DB1302_UNIT_03_STATION_CYCLE".SEQUENCE.GENERAL_CONDITIONS )
      I_Contact( "DB1302_UNIT_03_STATION_CYCLE".SEQUENCE.RUNNING )
      Coil( "DB1302_UNIT_03_STATION_CYCLE".SEQUENCE.GENERAL_CONDITIONS_HELP )
   END_RUNG
   // the same network as SCL:
   "DB1302_UNIT_03_STATION_CYCLE".SEQUENCE.GENERAL_CONDITIONS_HELP := NOT (NOT "DB1302_UNIT_03_STATION_CYCLE".SEQUENCE.SEMI_AUTO_REQUEST) AND NOT "DB1302_UNIT_03_STATION_CYCLE".SEQUENCE.GENERAL_CONDITIONS AND NOT "DB1302_UNIT_03_STATION_CYCLE".SEQUENCE.RUNNING;
END_REGION

REGION Network 20: INITIAL CONDITIONS HELP
   RUNG wire#powerrail
      I_Contact( "DB1302_UNIT_03_STATION_CYCLE".SEQUENCE.SEMI_AUTO_REQUEST )
      Not()
      Contact( "DB1302_UNIT_03_STATION_CYCLE".SEQUENCE.GENERAL_CONDITIONS )
      I_Contact( "DB1302_UNIT_03_STATION_CYCLE".SEQUENCE.RUNNING )
      I_Contact( "DB1302_UNIT_03_STATION_CYCLE".SEQUENCE.INITIAL_CONDITIONS )
      Coil( "DB1302_UNIT_03_STATION_CYCLE".SEQUENCE.INITIAL_CONDITIONS_HELP )
   END_RUNG
   // the same network as SCL:
   "DB1302_UNIT_03_STATION_CYCLE".SEQUENCE.INITIAL_CONDITIONS_HELP := NOT (NOT "DB1302_UNIT_03_STATION_CYCLE".SEQUENCE.SEMI_AUTO_REQUEST) AND "DB1302_UNIT_03_STATION_CYCLE".SEQUENCE.GENERAL_CONDITIONS AND NOT "DB1302_UNIT_03_STATION_CYCLE".SEQUENCE.RUNNING AND NOT "DB1302_UNIT_03_STATION_CYCLE".SEQUENCE.INITIAL_CONDITIONS;
END_REGION

REGION Network 21: HMI STATUS
   RUNG wire#powerrail
      I_Contact( "DB1302_UNIT_03_STATION_CYCLE".SEQUENCE.RUNNING )
      Coil( "DB505_HMI_SetUp".Setup1.Movement_EndPos.movement240EndPosRight )
   END_RUNG
   // the same network as SCL:
   "DB505_HMI_SetUp".Setup1.Movement_EndPos.movement240EndPosRight := NOT "DB1302_UNIT_03_STATION_CYCLE".SEQUENCE.RUNNING;
END_REGION

REGION Network 22: HMI STATUS
   RUNG wire#powerrail
      Contact( "DB2001_MODES_GENERAL".GENERAL.SEMIAUTO_SELECTED )
      Contact( "DB1302_UNIT_03_STATION_CYCLE".SEQUENCE.GENERAL_CONDITIONS )
      Contact( "DB1302_UNIT_03_STATION_CYCLE".SEQUENCE.INITIAL_CONDITIONS )
      Coil( "DB505_HMI_SetUp".Setup1.Movement_Executability.movement240ExecutabilityRight )
   END_RUNG
   // the same network as SCL:
   "DB505_HMI_SetUp".Setup1.Movement_Executability.movement240ExecutabilityRight := "DB2001_MODES_GENERAL".GENERAL.SEMIAUTO_SELECTED AND "DB1302_UNIT_03_STATION_CYCLE".SEQUENCE.GENERAL_CONDITIONS AND "DB1302_UNIT_03_STATION_CYCLE".SEQUENCE.INITIAL_CONDITIONS;
END_REGION

REGION Network 23: HMI STATUS
   RUNG wire#powerrail
      Contact( "DB1302_UNIT_03_STATION_CYCLE".SEQUENCE.RUNNING )
      Contact( "M_0.5_SEC_2HZ" )
      Coil( "DB505_HMI_SetUp".Setup1.MovementActive.movement240ActiveRight )
   END_RUNG
   // the same network as SCL:
   "DB505_HMI_SetUp".Setup1.MovementActive.movement240ActiveRight := "DB1302_UNIT_03_STATION_CYCLE".SEQUENCE.RUNNING AND "M_0.5_SEC_2HZ";
END_REGION
END_FUNCTION
